FUNCTION_BLOCK DAMPER_CTL (* Variable Air Volume Damper Controller *)
  (* Standard: 61499-1; ApplicationDomain: HVAC; Function: Control; Type: Variable Air Volume; Description: VAV Damper Controller *)
  (* Version 0.0, 2006-05-01, JHC, Holobloc Inc *)
  (* Compiler header: package fb.rt.hvac; *)
  (* Compiler Java Sun JDK 1.5.0 *)
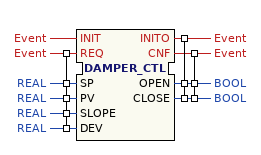
  EVENT_INPUT
    INIT; (* Initialization Request *)
    REQ WITH SP, PV, SLOPE, DEV; (* Periodic Execution Clock *)
  END_EVENT
  EVENT_OUTPUT
    INITO WITH OPEN, CLOSE; (* Initialization Confirm *)
    CNF WITH OPEN, CLOSE; (* OPEN/CLOSE command value change *)
  END_EVENT
  VAR_INPUT
    SP : REAL; (* Set point, fraction full scale *)
    PV : REAL; (* Estimated Velocity Sensor Reading, fraction full scale *)
    SLOPE : REAL; (* Slope of regressed PV, units per clock period. *)
    DEV : REAL; (* Estimated standard deviation from regression line *)
  END_VAR
  VAR_OUTPUT
    OPEN : BOOL; (* Damper OPEN command *)
    CLOSE : BOOL; (* Damper CLOSE command *)
  END_VAR
END_FUNCTION_BLOCK
